Fanuc KAREL source: IO0026.KL

-- PROVISIONAL review KL for V940-1; original PC SHA256 1f5e77bfa2e8bfea80e151975e6cb4313613ebf88bca2468bba0f8509a4d6b5c
-- Incomplete behavior may be omitted. Consult companion uncertainty JSON. Do not deploy.
PROGRAM IO0026
%NOLOCKGROUP
-- UNRESOLVED_LOCAL_POOL 5 cells at code offset 13; source declarations unknown
-- DIRECT_LOCAL_WORD_ACCESS alone does not prove INTEGER, REAL, or BOOLEAN
BEGIN
  -- V9_ZERO_TABLE_METADATA_HINT layout=0001; no indexed target words; source/name/runtime held
  -- V9_ZERO_GLOBAL_LAYOUT_HINT count-one $GROUP table, zero relocation slots, two routine descriptors; executable preamble and source held
  -- V9_SIGNAL_INDEX_HINT DOUT write index_cell=40
  -- UNRESOLVED_PC offsets 0-18; opcodes 2B,2C,7B
  -- UNRESOLVED_PC offsets 23-30; opcodes 9D,23
  -- UNRESOLVED_PC offsets 35-49; opcodes 2E,22,9D,33,35
  -- UNRESOLVED_PC offsets 54-61; opcodes 9D,23
  -- UNRESOLVED_PC offsets 66-77; opcodes 2E,23
  -- UNRESOLVED_PC offsets 82-96; opcodes 21,21,1A
  -- UNRESOLVED_PC offsets 101-105; opcodes 7F
  -- UNRESOLVED_PC offsets 110-114; opcodes 27,AA
  -- UNRESOLVED_PC offsets 119-123; opcodes 7F
END IO0026
